// TIA Portal V20 export
DATA_BLOCK "DB_ExtraMissingPart"   // DB113
// stored: InstanceOfName FB_ExtraMissingPart, InstanceOfType FB
"FB_ExtraMissingPart"
   // VAR
   //    sRT_UndrilledGripperClosedWithPart : R_TRIG;
   //    sRT_UndrilledGripperClosedWithoutPart { S7_SetPoint := 'True'} : R_TRIG;
   //    sRT_DrilledGripperClosedWithPart : R_TRIG;
   //    sRT_DrilledGripperClosedWithoutPart { S7_SetPoint := 'True'} : R_TRIG;
   //    sRT_FixturePartControlGood { S7_SetPoint := 'True'} : R_TRIG;
   //    sRT_FixturePartControlBad { S7_SetPoint := 'True'} : R_TRIG;
   //    sRT_UndrilledGripperOpen { S7_SetPoint := 'True'} : R_TRIG;
   //    sRT_DrilledGripperOpen { S7_SetPoint := 'True'} : R_TRIG;
   //    sTON_UndrilledGripperClosedWithPart { S7_SetPoint := 'True'} : TON_TIME;
   //    sTON_UndrilledGripperClosedWithoutPart { S7_SetPoint := 'True'} : TON_TIME;
   //    sTON_DrilledGripperClosedWithPart { S7_SetPoint := 'True'} : TON_TIME;
   //    sTON_DrilledGripperClosedWithoutPart { S7_SetPoint := 'True'} : TON_TIME;
   //    sTON_FixturePartControlGood { S7_SetPoint := 'True'} : TON_TIME;
   //    sTON_FixturePartControlBad { S7_SetPoint := 'True'} : TON_TIME;
   //    sTON_UndrilledGripperOpen { S7_SetPoint := 'True'} : TON_TIME;
   //    sTON_DrilledGripperOpen { S7_SetPoint := 'True'} : TON_TIME;
   //    sExtraPartUndrilledGripper { S7_SetPoint := 'True'} : Bool;
   //    sExtraPartDrilledGripper : Bool;
   //    sMissingPartUndrilledGripper { S7_SetPoint := 'True'} : Bool;
   //    sMissingPartDrilledGripper : Bool;
   //    sExtraPartFixture : Bool;
   //    sMissingPartFixture : Bool;
   //    sGlobalExtraMissing : Bool;
   //    sUndrilledGripperClosedWithPart : Bool;
   //    sUndrilledGripperClosedWithoutPart { S7_SetPoint := 'True'} : Bool;
   //    sDrilledGripperClosedWithPart : Bool;
   //    sDrilledGripperClosedWithoutPart { S7_SetPoint := 'True'} : Bool;
   //    sFixturePartControlGood { S7_SetPoint := 'True'} : Bool;
   //    sFixturePartControlBad { S7_SetPoint := 'True'} : Bool;
   //    sUndrilledGripperOpen { S7_SetPoint := 'True'} : Bool;
   //    sDrilledGripperOpen { S7_SetPoint := 'True'} : Bool;
   // END_VAR
BEGIN
END_DATA_BLOCK
